# B&R Automation Studio project Panasonic_LinkaPowerCP2_A2021055 (part 3)

### Config.mprecipexml - 5PC900_TS17_00/mappServices/Config.mprecipexml
```
Element gRemPremenneP1 (Type=mprecipexml)
```

### Config_1.mprecipexml - 5PC900_TS17_00/mappServices/Config_1.mprecipexml
```
Element gRemPremenneP2 (Type=mprecipexml)
```

### Config_2.mprecipexml - 5PC900_TS17_00/mappServices/Config_2.mprecipexml
```
Element gRemPremenneP34 (Type=mprecipexml)
```

### Config_3.mpalarmxhistory - 5PC900_TS17_00/mappServices/Config_3.mpalarmxhistory
```
Element gAlarmXHistory (Type=mpalarmxhistory)
  mapp.AlarmX.History:
    Export:
      FileNamePattern = Alarms_%d_%m_%Y_%H_%M_%S.csv
      TimeStampPattern = %d-%m-%Y %H:%M:%S:%L
```

### Config_4.mpalarmxcore - 5PC900_TS17_00/mappServices/Config_4.mpalarmxcore
```
Element gAlarmXCore (Type=mpalarmxcore)
  mapp.AlarmX.Core.Configuration:
    [0]:
      Name = A100
      Message = ST1_Vytah - paletka na vystupe dopravnika vytahu !!!
      Code = 100
      Behavior = PersistentAlarm
    [1]:
      Name = A101
      Message = ST1_Vytah - narusenie optickej bariery !!!
      Code = 101
      Behavior = PersistentAlarm
    [2]:
      Name = A102
      Message = ST1_Vytah - porucha navezenia paletky na dopravnik vytahu !!!
      Code = 102
      Behavior = PersistentAlarm
    [3]:
      Name = A103
      Message = ST1_Vytah - porucha precitania kodu paletky !!!
      Code = 103
      Behavior = PersistentAlarm
    [4]:
      Name = A104
      Message = ST1_Vytah - porucha komunikacie zo serverom !!!
      Code = 104
      Behavior = PersistentAlarm
    [5]:
      Name = A105
      Message = ST1_Vytah - porucha odoslania fotiek na server !!!
      Code = 105
      Behavior = PersistentAlarm
    [6]:
      Name = A106
      Message = ST1_Vytah - CAM 2 porucha komunikacie FTP !!!
      Code = 106
      Behavior = PersistentAlarm
    [7]:
      Name = A107
      Message = ST1_Vytah - CAM 3 porucha komunikacie FTP !!!
      Code = 107
      Behavior = PersistentAlarm
    [8]:
      Name = A108
      Message = ST1_Vytah - CAM 4 porucha komunikacie FTP !!!
      Code = 108
      Behavior = PersistentAlarm
    [9]:
      Name = A109
      Message = ST1_Vytah - CAM 5 porucha komunikacie FTP !!!
      Code = 109
      Behavior = PersistentAlarm
    [10]:
      Name = A110
      Message = ST1_Vytah - porucha serva zdvihu vytahu !!!
      Code = 110
      Behavior = PersistentAlarm
    [11]:
      Name = A111
      Message = ST2_Srobovanie - porucha vysunutia centrovacky !!!
      Code = 111
      Behavior = PersistentAlarm
    [12]:
      Name = A112
      Message = ST2_Srobovanie - porucha zasunutia centrovacky !!!
      Code = 112
      Behavior = PersistentAlarm
    [13]:
      Name = A113
      Message = ST2_Srobovanie - porucha precitania kodu paletky !!!
      Code = 113
      Behavior = PersistentAlarm
    [14]:
      Name = A114
      Message = ST2_Srobovanie - porucha komunikacie zo serverom !!!
      Code = 114
      Behavior = PersistentAlarm
    [15]:
      Name = A115
      Message = ST2_Srobovanie - porucha odoslania fotiek na server !!!
      Code = 115
      Behavior = PersistentAlarm
    [16]:
      Name = A116
      Message = ST2_Srobovanie - CAM 6 porucha komunikacie FTP !!!
      Code = 116
      Behavior = PersistentAlarm
    [17]:
      Name = A117
      Message = ST2_Srobovanie - porucha serva manipulatora os X !!!
      Code = 117
      Behavior = PersistentAlarm
    [18]:
      Name = A118
      Message = ST2_Srobovanie - porucha serva manipulatora os Y !!!
      Code = 118
      Behavior = PersistentAlarm
    [19]:
      Name = A119
      Message = ST2_Srobovanie - skrutka K30 nieje pripravena !!!
      Code = 119
      Behavior = PersistentAlarm
    [20]:
      Name = A120
      Message = ST2_Srobovanie - skrutka M5 nieje pripravena !!!
      Code = 120
      Behavior = PersistentAlarm
    [21]:
      Name = A121
      Message = ST2_Srobovanie - skrutka M4 nieje pripravena !!!
      Code = 121
      Behavior = PersistentAlarm
    [22]:
      Name = A122
      Message = P1_Robot - porucha napajania !!!
      Code = 122
      Behavior = PersistentAlarm
    [23]:
      Name = A123
      Message = P1_Robot - nieje online !!!
      Code = 123
      Behavior = PersistentAlarm
    [24]:
      Name = A124
      Message = Pracovisko 1 - Porucha tlaku vzduchu !!!
      Code = 124
      Behavior = PersistentAlarm
    [25]:
      Name = A125
      Message = Pracovisko 1 - Moduly IO niesu online !!!
      Code = 125
      Behavior = PersistentAlarm
    [26]:
      Name = A126
      Message = ST2_Srobovanie - porucha serva manipulatora os Z M4 !!!
      Code = 126
      Behavior = PersistentAlarm
    [27]:
      Name = A127
      Message = ST2_Srobovanie - porucha serva manipulatora os Z M5 !!!
      Code = 127
      Behavior = PersistentAlarm
    [28]:
      Name = A128
      Message = Pracovisko 1 - Porucha skrutkovacieho setu M4 !!!
      Code = 128
      Behavior = PersistentAlarm
    [29]:
      Name = A129
      Message = Pracovisko 1 - Porucha skrutkovacieho setu M5 !!!
      Code = 129
      Behavior = PersistentAlarm
    [30]:
      Name = A130
      Message = Pracovisko 1 - Narusenie optickej bariery na vystupe bunky !!!
      Code = 130
      Behavior = PersistentAlarm
    [31]:
      Name = A131
      Message = Pracovisko 1 - Modul DS12 nieje online !!!
      Code = 131
      Behavior = PersistentAlarm
    [32]:
      Name = A132
      Message = Pracovisko 1 - Modul SI11 nieje online !!!
      Code = 132
      Behavior = PersistentAlarm
    [33]:
      Name = A133
      Message = Pracovisko 1 - Modul SI12 nieje online !!!
      Code = 133
      Behavior = PersistentAlarm
    [34]:
      Name = A134
      Message = Pracovisko 1 - Ventilovy termnal Bunky 1 nieje online !!!
      Code = 134
      Behavior = PersistentAlarm
    [35]:
      Name = A135
      Message = Pracovisko 1 - Ventilovy termnal VT5 nieje online !!!
      Code = 135
      Behavior = PersistentAlarm
    [36]:
      Name = A136
      Message = ST2_Srobovanie - Skrutkovacka K30 nieje online !!!
      Code = 136
      Behavior = PersistentAlarm
    [37]:
      Name = A137
      Message = ST2_Srobovanie - Skrutkovacka M5 nieje online !!!
      Code = 137
      Behavior = PersistentAlarm
    [38]:
      Name = A138
      Message = ST2_Srobovanie - Skrutkovacka M4 nieje online !!!
      Code = 138
      Behavior = PersistentAlarm
    [39]:
      Name = A139
      Message = Pracovisko 1 - Kamery KAM2, KAM4 a KAM6 niesu online !!!
      Code = 139
      Behavior = PersistentAlarm
    [40]:
      Name = A140
      Message = Pracovisko 1 - Kamera KAM3 nieje online !!!
      Code = 140
      Behavior = PersistentAlarm
    [41]:
      Name = A141
      Message = Pracovisko 1 - Kamera KAM5 nieje online !!!
      Code = 141
      Behavior = PersistentAlarm
    [42]:
      Name = A142
      Message = ST2_Srobovanie - Porucha vysunutia skrutkovacky K30 !!!
      Code = 142
      Behavior = PersistentAlarm
    [43]:
      Name = A143
      Message = ST2_Srobovanie - Porucha vysunutia skrutkovacky M5  !!!
      Code = 143
      Behavior = PersistentAlarm
    [44]:
      Name = A144
      Message = ST2_Srobovanie - Porucha vysunutia skrutkovacky M4 !!!
      Code = 144
      Behavior = PersistentAlarm
    [45]:
      Name = A145
      Message = P1_Robot - porucha !!!
      Code = 145
      Behavior = PersistentAlarm
    [46]:
      Name = A146
      Message = ST2_Srobovanie - Presiahnuty cas skrutkovania skrutky K30 !!!
      Code = 146
      Behavior = PersistentAlarm
    [47]:
      Name = A147
      Message = ST2_Srobovanie - Presiahnuty cas skrutkovania skrutky M5 !!!
      Code = 147
      Behavior = PersistentAlarm
    [48]:
      Name = A148
      Message = ST2_Srobovanie - Presiahnuty cas skrutkovania skrutky M4 !!!
      Code = 148
      Behavior = PersistentAlarm
    [49]:
      Name = A149
      Message = ST2_Srobovanie - Skrutkovacka K30 nieje READY !!!
      Code = 149
      Behavior = PersistentAlarm
    [50]:
      Name = A150
      Message = ST2_Srobovanie - Skrutkovacka M5 nieje READY !!!
      Code = 150
      Behavior = PersistentAlarm
    [51]:
      Name = A151
      Message = ST2_Srobovanie - Skrutkovacka M4 nieje READY !!!
      Code = 151
      Behavior = PersistentAlarm
    [52]:
      Name = A152
      Message = Pracovisko 1 - Prekrocena teplota motora vrchneho dopravnika !!!
      Code = 152
      Behavior = PersistentAlarm
    [53]:
      Name = A153
      Message = Pracovisko 1 - Prekrocena teplota motora spodneho dopravnika !!!
      Code = 153
      Behavior = PersistentAlarm
    [54]:
      Name = A154
      Message = Pracovisko 1 - Narusenie optickej bariery na vstupe bunky !!!
      Code = 154
      Behavior = PersistentAlarm
    [55]:
      Name = A155
      Message = ST1_Vytah - Prekrocena teplota motora dopravnika !!!
      Code = 155
      Behavior = PersistentAlarm
    [56]:
      Name = A156
      Message = Pracovisko 1 - Bolo stlacene tlacitko CS na ovladacom paneli !!!
      Code = 156
      Behavior = PersistentAlarm
    [57]:
      Name = A157
      Message = Pracovisko 1 - Bolo stlacene tlacitko CS na rozvodnej skrini !!!
      Code = 157
      Behavior = PersistentAlarm
    [58]:
      Name = A158
      Message = Pracovisko 1 - Bolo stlacene tlacitko CS robota !!!
      Code = 158
      Behavior = PersistentAlarm
    [59]:
      Name = A159
      Message = P1_Robot - Porucha odobratia foamov z paletky !!!
      Code = 159
      Behavior = PersistentAlarm
    [60]:
      Name = A160
      Message = P1_Robot - Porucha odobratia busbarov z paletky !!!
      Code = 160
      Behavior = PersistentAlarm
    [61]:
      Name = A161
      Message = ST2_Srobovanie - Porucha vyvezenia paletky zo stopra !!!
      Code = 161
      Behavior = PersistentAlarm
    [62]:
      Name = A162
      Message = P1_Akumulacny stoper - Porucha vyvezenia paletky zo stopra !!!
      Code = 162
      Behavior = PersistentAlarm
    [63]:
      Name = A163
      Message = P1_Spodny stoper - Porucha vyvezenia paletky zo stopra !!!
      Code = 163
      Behavior = PersistentAlarm
    [64]:
      Name = A164
      Message = ST1_Vytah - Porucha komunikacie s kamerou CAM 2 !!!
      Code = 164
      Behavior = PersistentAlarm
    [65]:
      Name = A165
      Message = ST1_Vytah - Porucha komunikacie s kamerou CAM 5 !!!
      Code = 165
      Behavior = PersistentAlarm
    [66]:
      Name = A166
      Message = ST1_Vytah - Porucha komunikacie s kamerou CAM 4 !!!
      Code = 166
      Behavior = PersistentAlarm
    [67]:
      Name = A167
      Message = ST1_Vytah - Porucha komunikacie s kamerou CAM 3 !!!
      Code = 167
      Behavior = PersistentAlarm
    [68]:
      Name = A168
      Message = ST2_Srobovanie - Porucha komunikacie s kamerou CAM 6 !!!
      Code = 168
      Behavior = PersistentAlarm
    [69]:
      Name = A200
      Message = ST3_Zakladanie tesnenia - porucha precitania kodu paletky !!!
      Code = 200
      Behavior = PersistentAlarm
    [70]:
      Name = A201
      Message = ST3_Zakladanie tesnenia - porucha precitania QR kodu !!!
      Code = 201
      Behavior = PersistentAlarm
    [71]:
      Name = A202
      Message = ST3_Zakladanie tesnenia - porucha serva zdvihu !!!
      Code = 202
      Behavior = PersistentAlarm
    [72]:
      Name = A203
      Message = ST3_Zakladanie tesnenia - porucha serva pojazdu !!!
      Code = 203
      Behavior = PersistentAlarm
    [73]:
      Name = A204
      Message = ST3_Zakladanie tesnenia - porucha vysunutia pritlacania !!!
      Code = 204
      Behavior = PersistentAlarm
    [74]:
      Name = A205
      Message = ST3_Zakladanie tesnenia - porucha zasunutia pritlacania !!!
      Code = 205
      Behavior = PersistentAlarm
    [75]:
      Name = A206
      Message = ST3_Zakladanie tesnenia - narusenie optickej bariery !!!
      Code = 206
      Behavior = PersistentAlarm
    [76]:
      Name = A207
      Message = ST3_Zakladanie tesnenia - bol stlaceny bumper suflika !!!
      Code = 207
      Behavior = PersistentAlarm
    [77]:
      Name = A208
      Message = ST3_Zakladanie tesnenia - porucha snimaca kopita IS7 !!!
      Code = 208
      Behavior = PersistentAlarm
    [78]:
      Name = A209
      Message = ST4_Maticovacka - porucha vysunutia centrovacky !!!
      Code = 209
      Behavior = PersistentAlarm
    [79]:
      Name = A210
      Message = ST4_Maticovacka - porucha zasunutia centrovacky !!!
      Code = 210
      Behavior = PersistentAlarm
    [80]:
      Name = A211
      Message = ST4_Maticovacka - porucha precitania kodu paletky !!!
      Code = 211
      Behavior = PersistentAlarm
    [81]:
      Name = A212
      Message = ST5_Srobovanie - porucha vysunutia centrovacky !!!
      Code = 212
      Behavior = PersistentAlarm
    [82]:
      Name = A213
      Message = ST5_Srobovanie - porucha zasunutia centrovacky !!!
      Code = 213
      Behavior = PersistentAlarm
    [83]:
      Name = A214
      Message = ST5_Srobovanie - porucha precitania kodu paletky !!!
      Code = 214
      Behavior = PersistentAlarm
    [84]:
      Name = A215
      Message = ST5_Srobovanie - porucha serva manipulatora os X !!!
      Code = 215
      Behavior = PersistentAlarm
    [85]:
      Name = A216
      Message = ST5_Srobovanie - porucha serva manipulatora os Y !!!
      Code = 216
      Behavior = PersistentAlarm
    [86]:
      Name = A217
      Message = ST6_Zvaranie - porucha vysunutia centrovacky !!!
      Code = 217
      Behavior = PersistentAlarm
    [87]:
      Name = A218
      Message = ST6_Zvaranie - porucha zasunutia centrovacky !!!
      Code = 218
      Behavior = PersistentAlarm
    [88]:
      Name = A219
      Message = ST6_Zvaranie - porucha precitania kodu paletky !!!
      Code = 219
      Behavior = PersistentAlarm
    [89]:
      Name = A220
      Message = ST6_Zvaranie - porucha serva zdvihu zvarania !!!
      Code = 220
      Behavior = PersistentAlarm
    [90]:
      Name = A221
      Message = ST6_Zvaranie - porucha presunu pojazdu zvarania !!!
      Code = 221
      Behavior = PersistentAlarm
    [91]:
      Name = A222
      Message = ST6_Zvaranie - porucha zvaracky !!!
      Code = 222
      Behavior = PersistentAlarm
    [92]:
      Name = A223
      Message = ST6_Cistenie - porucha zatvorenia dveri !!!
      Code = 223
      Behavior = PersistentAlarm
    [93]:
      Name = A224
      Message = ST6_Cistenie - porucha otvorenia dveri !!!
      Code = 224
      Behavior = PersistentAlarm
    [94]:
      Name = A225
      Message = ST3_Zakladanie tesnenia - CAM 1 porucha komunikacie FTP !!!
      Code = 225
      Behavior = PersistentAlarm
    [95]:
      Name = A226
      Message = ST3_Zakladanie tesnenia - CAM 7 porucha komunikacie FTP !!!
      Code = 226
      Behavior = PersistentAlarm
    [96]:
      Name = A227
      Message = ST3_Zakladanie tesnenia - CAM 8 porucha komunikacie FTP !!!
      Code = 227
      Behavior = PersistentAlarm
    [97]:
      Name = A228
      Message = ST3_Zakladanie tesnenia - CAM 17 porucha komunikacie FTP !!!
      Code = 228
      Behavior = PersistentAlarm
    [98]:
      Name = A229
      Message = ST4_Maticovacka - CAM 9 porucha komunikacie FTP !!!
      Code = 229
      Behavior = PersistentAlarm
    [99]:
      Name = A230
      Message = ST3_Zakladanie tesnenia - porucha komunikacie zo serverom !!!
      Code = 230
      Behavior = PersistentAlarm
    [100]:
      Name = A231
      Message = ST4_Maticovacka - porucha komunikacie zo serverom !!!
      Code = 231
      Behavior = PersistentAlarm
    [101]:
      Name = A232
      Message = ST5_Srobovanie - CAM 10 porucha komunikacie FTP !!!
      Code = 232
      Behavior = PersistentAlarm
    [102]:
      Name = A233
      Message = ST5_Srobovanie - porucha komunikacie zo serverom !!!
      Code = 233
      Behavior = PersistentAlarm
    [103]:
      Name = A234
      Message = ST6_Zvaranie - CAM 11 porucha komunikacie FTP !!!
      Code = 234
      Behavior = PersistentAlarm
    [104]:
      Name = A235
      Message = ST6_Zvaranie - CAM 12 porucha komunikacie FTP !!!
      Code = 235
      Behavior = PersistentAlarm
    [105]:
      Name = A236
      Message = ST6_Zvaranie - porucha komunikacie zo serverom !!!
      Code = 236
      Behavior = PersistentAlarm
    [106]:
      Name = A237
      Message = ST5_Srobovanie - skrutka M4 nieje pripravena !!!
      Code = 237
      Behavior = PersistentAlarm
    [107]:
      Name = A238
      Message = ST5_Srobovanie - skrutka M5 nieje pripravena !!!
      Code = 238
      Behavior = PersistentAlarm
    [108]:
      Name = A239
      Message = ST5_Srobovanie - skrutka M6 nieje pripravena !!!
      Code = 239
      Behavior = PersistentAlarm
    [109]:
      Name = A240
      Message = ST4_Maticovacka - matica M4 nieje pripravena !!!
      Code = 240
      Behavior = PersistentAlarm
    [110]:
      Name = A241
      Message = ST5_Srobovanie - porucha serva manipulatora os X !!!
      Code = 241
      Behavior = PersistentAlarm
    [111]:
      Name = A242
      Message = ST5_Srobovanie - porucha serva manipulatora os Y !!!
      Code = 242
      Behavior = PersistentAlarm
    [112]:
      Name = A243
      Message = P2_Robot - porucha napajania !!!
      Code = 243
      Behavior = PersistentAlarm
    [113]:
      Name = A244
      Message = P2_Robot - nieje online !!!
      Code = 244
      Behavior = PersistentAlarm
    [114]:
      Name = A245
      Message = Pracovisko 2 - Porucha tlaku vzduchu !!!
      Code = 245
      Behavior = PersistentAlarm
    [115]:
      Name = A246
      Message = Pracovisko 2 - Moduly IO niesu online !!!
      Code = 246
      Behavior = PersistentAlarm
    [116]:
      Name = A247
      Message = ST5_Srobovanie - porucha serva manipulatora os Z M4 !!!
      Code = 247
      Behavior = PersistentAlarm
    [117]:
      Name = A248
      Message = Pracovisko 2 - Porucha skrutkovacieho setu M4 !!!
      Code = 248
      Behavior = PersistentAlarm
    [118]:
      Name = A249
      Message = Pracovisko 2 - Porucha skrutkovacieho setu matice M4 !!!
      Code = 249
    [119]:
      Name = A250
      Message = Pracovisko 2 - Porucha komunikacie s Panatrace !!!
      Code = 250
      Behavior = PersistentAlarm
    [120]:
      Name = A251
      Message = Pracovisko 2 - Modul DM21 nieje online !!!
      Code = 251
    [121]:
      Name = A252
      Message = Pracovisko 2 - Modul DS21 nieje online !!!
      Code = 252
      Behavior = PersistentAlarm
    [122]:
      Name = A253
      Message = Pracovisko 2 - Modul DS22 nieje online !!!
      Code = 253
      Behavior = PersistentAlarm
    [123]:
      Name = A254
      Message = Pracovisko 2 - Modul DS23 nieje online !!!
      Code = 254
      Behavior = PersistentAlarm
    [124]:
      Name = A255
      Message = Pracovisko 2 - Modul SI21 nieje online !!!
      Code = 255
      Behavior = PersistentAlarm
    [125]:
      Name = A256
      Message = Pracovisko 2 - Modul SI22 nieje online !!!
      Code = 256
      Behavior = PersistentAlarm
    [126]:
      Name = A257
      Message = Pracovisko 2 - Ventilovy termnal Bunky 2 nieje online !!!
      Code = 257
      Behavior = PersistentAlarm
    [127]:
      Name = A258
      Message = Pracovisko 2 - Ventilovy termnal VT2 nieje online !!!
      Code = 258
      Behavior = PersistentAlarm
    [128]:
      Name = A259
      Message = Pracovisko 2 - Ventilovy termnal VT3 nieje online !!!
      Code = 259
      Behavior = PersistentAlarm
    [129]:
      Name = A260
      Message = ST5_Srobovanie - Skrutkovacka M4 nieje online !!!
      Code = 260
      Behavior = PersistentAlarm
    [130]:
      Name = A261
      Message = ST5_Srobovanie - Skrutkovacka M5 nieje online !!!
      Code = 261
      Behavior = PersistentAlarm
    [131]:
      Name = A262
      Message = ST5_Srobovanie - Skrutkovacka M6 nieje online !!!
      Code = 262
      Behavior = PersistentAlarm
    [132]:
      Name = A263
      Message = ST4_Maticovacka - Maticovacka M4 nieje online !!!
      Code = 263
      Behavior = PersistentAlarm
    [133]:
      Name = A264
      Message = Pracovisko 2 - Kamery KAM1, KAM7, KAM10, KAM11, KAM12 a KAM17 niesu online !!!
      Code = 264
      Behavior = PersistentAlarm
    [134]:
      Name = A265
      Message = Pracovisko 2 - Kamera KAM8 nieje online !!!
      Code = 265
      Behavior = PersistentAlarm
    [135]:
      Name = A266
      Message = Pracovisko 2 - Kamera KAM9 nieje online !!!
      Code = 266
      Behavior = PersistentAlarm
    [136]:
      Name = A267
      Message = ST4_Maticovacka - Porucha maticovacky M4 !!!
      Code = 267
      Behavior = PersistentAlarm
    [137]:
      Name = A268
      Message = ST5_Srobovanie - Porucha vysunutia skrutkovacky M4 !!!
      Code = 268
      Behavior = PersistentAlarm
    [138]:
      Name = A269
      Message = ST5_Srobovanie - Porucha vysunutia skrutkovacky M5 !!!
      Code = 269
      Behavior = PersistentAlarm
    [139]:
      Name = A270
      Message = ST5_Srobovanie - Porucha vysunutia skrutkovacky M6 !!!
      Code = 270
      Behavior = PersistentAlarm
    [140]:
      Name = A271
      Message = P2_Robot - porucha !!!
      Code = 271
      Behavior = PersistentAlarm
    [141]:
      Name = A272
      Message = ST5_Srobovanie - Presiahnuty cas skrutkovania skrutky M4 !!!
      Code = 272
      Behavior = PersistentAlarm
    [142]:
      Name = A273
      Message = ST5_Srobovanie - Presiahnuty cas skrutkovania skrutky M5 !!!
      Code = 273
      Behavior = PersistentAlarm
    [143]:
      Name = A274
      Message = ST5_Srobovanie - Presiahnuty cas skrutkovania skrutky M6 !!!
      Code = 274
      Behavior = PersistentAlarm
    [144]:
      Name = A275
      Message = ST5_Srobovanie - Skrutkovacka M4 nieje READY !!!
      Code = 275
      Behavior = PersistentAlarm
    [145]:
      Name = A276
      Message = ST5_Srobovanie - Skrutkovacka M5 nieje READY !!!
      Code = 276
      Behavior = PersistentAlarm
    [146]:
      Name = A277
      Message = ST5_Srobovanie - Skrutkovacka M6 nieje READY !!!
      Code = 277
      Behavior = PersistentAlarm
    [147]:
      Name = A278
      Message = Pracovisko 2 - Prekrocena teplota motora vrchneho dopravnika !!!
      Code = 278
      Behavior = PersistentAlarm
    [148]:
      Name = A279
      Message = Pracovisko 2 - Prekrocena teplota motora spodneho dopravnika !!!
      Code = 279
      Behavior = PersistentAlarm
    [149]:
      Name = A280
      Message = Pracovisko 2 - Narusenie optickej bariery na vystupe !!!
      Code = 280
      Behavior = PersistentAlarm
    [150]:
      Name = A281
      Message = Pracovisko 2 - Bolo stlacene tlacitko CS na ovladacom paneli !!!
      Code = 281
      Behavior = PersistentAlarm
    [151]:
      Name = A282
      Message = Pracovisko 2 - Bolo stlacene tlacitko CS na rozvodnej skrini !!!
      Code = 282
      Behavior = PersistentAlarm
    [152]:
      Name = A283
      Message = Pracovisko 2 - Bolo stlacene tlacitko CS robota !!!
      Code = 283
      Behavior = PersistentAlarm
    [153]:
      Name = A284
      Message = Pracovisko 2 - Bolo stlacene tlacitko CS na dvojrucnom ovladani !!!
      Code = 284
      Behavior = PersistentAlarm
    [154]:
      Name = A285
      Message = P2_Robot - Porucha odobratia Top Coveru z paletky !!!
      Code = 285
      Behavior = PersistentAlarm
    [155]:
      Name = A286
      Message = ST3_Zakladanie tesnenia - Porucha vyvezenia paletky zo stopra !!!
      Code = 286
      Behavior = PersistentAlarm
    [156]:
      Name = A287
      Message = ST4_Maticovacka - Porucha vyvezenia paletky zo stopra !!!
      Code = 287
      Behavior = PersistentAlarm
    [157]:
      Name = A288
      Message = ST5_Srobovanie - Porucha vyvezenia paletky zo stopra !!!
      Code = 288
      Behavior = PersistentAlarm
    [158]:
      Name = A289
      Message = ST6_Zvaranie - Porucha vyvezenia paletky zo stopra !!!
      Code = 289
      Behavior = PersistentAlarm
    [159]:
      Name = A290
      Message = ST3_Zakladanie tesnenia - Porucha komunikacie s kamerou CAM 1 !!!
      Code = 290
    [160]:
      Name = A291
      Message = ST3_Zakladanie tesnenia - Porucha komunikacie s kamerou CAM 7 !!!
      Code = 291
      Behavior = PersistentAlarm
    [161]:
      Name = A292
      Message = ST3_Zakladanie tesnenia - Porucha komunikacie s kamerou CAM 8 !!!
      Code = 292
      Behavior = PersistentAlarm
    [162]:
      Name = A293
      Message = ST3_Zakladanie tesnenia - Porucha komunikacie s kamerou CAM 17 !!!
      Code = 293
      Behavior = PersistentAlarm
    [163]:
      Name = A294
      Message = ST4_Maticovacka - Porucha komunikacie s kamerou CAM 9 !!!
      Code = 294
      Behavior = PersistentAlarm
    [164]:
      Name = A295
      Message = ST5_Srobovanie - Porucha komunikacie s kamerou CAM 10 !!!
      Code = 295
      Behavior = PersistentAlarm
    [165]:
      Name = A296
      Message = ST6_Zvaranie - Porucha komunikacie s kamerou CAM 11 !!!
      Code = 296
      Behavior = PersistentAlarm
    [166]:
      Name = A297
      Message = ST6_Zvaranie - Porucha komunikacie s kamerou CAM 12 !!!
      Code = 297
      Behavior = PersistentAlarm
    [167]:
      Name = A298
      Message = ST4_Maticovacka - Porucha pripravy matice M4 !!!
      Code = 298
      Behavior = PersistentAlarm
    [168]:
      Name = A299
      Message = Akumulacny stoper - Porucha vyvezenia paletky zo stopra !!!
      Code = 299
      Behavior = PersistentAlarm
    [169]:
      Name = A300
      Message = ST7_Srobovanie - porucha vysunutia centrovacky !!!
      Code = 300
      Behavior = PersistentAlarm
    [170]:
      Name = A301
      Message = ST7_Srobovanie - porucha zasunutia centrovacky !!!
      Code = 301
      Behavior = PersistentAlarm
    [171]:
      Name = A302
      Message = ST8A_Leakage test A - porucha vysunutia centrovacky !!!
      Code = 302
      Behavior = PersistentAlarm
    [172]:
      Name = A303
      Message = ST8A_Leakage test A - porucha zasunutia centrovacky !!!
      Code = 303
      Behavior = PersistentAlarm
    [173]:
      Name = A304
      Message = ST8B_Leakage test B - porucha vysunutia centrovacky !!!
      Code = 304
      Behavior = PersistentAlarm
    [174]:
      Name = A305
      Message = ST8B_Leakage test B - porucha zasunutia centrovacky !!!
      Code = 305
      Behavior = PersistentAlarm
    [175]:
      Name = A306
      Message = ST8A_Leakage test A - porucha vysunutia pritlaku !!!
      Code = 306
      Behavior = PersistentAlarm
    [176]:
      Name = A307
      Message = ST8A_Leakage test A - porucha zasunutia pritlaku !!!
      Code = 307
      Behavior = PersistentAlarm
    [177]:
      Name = A308
      Message = ST8B_Leakage test B - porucha vysunutia pritlaku !!!
      Code = 308
      Behavior = PersistentAlarm
    [178]:
      Name = A309
      Message = ST8B_Leakage test B - porucha zasunutia pritlaku !!!
      Code = 309
      Behavior = PersistentAlarm
    [179]:
      Name = A310
      Message = ST8A_Leakage test A - porucha precitania kodu paletky !!!
      Code = 310
      Behavior = PersistentAlarm
    [180]:
      Name = A311
      Message = ST8A_Leakage test A - porucha komunikacie zo serverom !!!
      Code = 311
      Behavior = PersistentAlarm
    [181]:
      Name = A312
      Message = ST8B_Leakage test B - porucha precitania kodu paletky !!!
      Code = 312
      Behavior = PersistentAlarm
    [182]:
      Name = A313
      Message = ST8B_Leakage test B - porucha komunikacie zo serverom !!!
      Code = 313
      Behavior = PersistentAlarm
    [183]:
      Name = A314
      Message = ST8A_Leakage test A - je zalozeny nespravny typ spodneho kopita !!!
      Code = 314
      Behavior = PersistentAlarm
    [184]:
      Name = A315
      Message = ST8B_Leakage test B - je zalozeny nespravny typ spodneho kopita !!!
      Code = 315
      Behavior = PersistentAlarm
    [185]:
      Name = A316
      Message = ST7_Srobovanie - porucha vysunutia kontaktov HV testu !!!
      Code = 316
      Behavior = PersistentAlarm
    [186]:
      Name = A317
      Message = ST7_Srobovanie - porucha zasunutia kontaktov HV testu !!!
      Code = 317
      Behavior = PersistentAlarm
    [187]:
      Name = A318
      Message = ST7_Srobovanie - porucha vysunutia HV testu !!!
      Code = 318
      Behavior = PersistentAlarm
    [188]:
      Name = A319
      Message = ST7_Srobovanie - porucha zasunutia HV testu !!!
      Code = 319
      Behavior = PersistentAlarm
    [189]:
      Name = A320
      Message = ST7_Srobovanie - CAM 13 porucha komunikacie FTP !!!
      Code = 320
      Behavior = PersistentAlarm
    [190]:
      Name = A321
      Message = ST7_Srobovanie - porucha precitania kodu paletky !!!
      Code = 321
      Behavior = PersistentAlarm
    [191]:
      Name = A322
      Message = ST7_Srobovanie - porucha serva manipulatora os Y !!!
      Code = 322
      Behavior = PersistentAlarm
    [192]:
      Name = A323
      Message = Pracovisko 3 - Porucha tlaku vzduchu !!!
      Code = 323
      Behavior = PersistentAlarm
    [193]:
      Name = A324
      Message = ST7_Srobovanie - Skrutkovacka M5 nieje online !!!
      Code = 324
      Behavior = PersistentAlarm
    [194]:
      Name = A325
      Message = ST7_Srobovanie - porucha komunikacie zo serverom !!!
      Code = 325
      Behavior = PersistentAlarm
    [195]:
      Name = A326
      Message = ST7_HV Test - je zalozeny nespravny typ spodneho kopita !!!
      Code = 326
      Behavior = PersistentAlarm
    [196]:
      Name = A327
      Message = ST7_Srobovanie - skrutka M5 nieje pripravena !!!
      Code = 327
      Behavior = PersistentAlarm
    [197]:
      Name = A328
      Message = ST7_Srobovanie - skrutka K40 nieje pripravena !!!
      Code = 328
      Behavior = PersistentAlarm
    [198]:
      Name = A329
      Message = ST7_Srobovanie - Skrutkovacka K40 nieje online !!!
      Code = 329
      Behavior = PersistentAlarm
    [199]:
      Name = A330
      Message = ST7_Srobovanie - Kamera KAM13 nieje online !!!
      Code = 330
      Behavior = PersistentAlarm
    [200]:
      Name = A331
      Message = Pracovisko 3 - Moduly IO niesu online !!!
      Code = 331
      Behavior = PersistentAlarm
    [201]:
      Name = A332
      Message = ST7_Srobovanie - porucha serva manipulatora os Z M5 !!!
      Code = 332
      Behavior = PersistentAlarm
    [202]:
      Name = A333
      Message = Pracovisko 3 - Modul DI33 nieje online !!!
      Code = 333
      Behavior = PersistentAlarm
    [203]:
      Name = A334
      Message = Pracovisko 3 - Porucha skrutkovacieho setu M5 !!!
      Code = 334
      Behavior = PersistentAlarm
    [204]:
      Name = A335
      Message = Pracovisko 3 - Prekrocena teplota motora zadneho vrchneho dopravnika !!!
      Code = 335
      Behavior = PersistentAlarm
    [205]:
      Name = A336
      Message = Pracovisko 3 - Prekrocena teplota motora prveho priecneho dopravnika !!!
      Code = 336
      Behavior = PersistentAlarm
    [206]:
      Name = A337
      Message = Pracovisko 3 - Prekrocena teplota motora druheho priecneho dopravnika !!!
      Code = 337
      Behavior = PersistentAlarm
    [207]:
      Name = A338
      Message = Pracovisko 3 - Modul DS33 nieje online !!!
      Code = 338
      Behavior = PersistentAlarm
    [208]:
      Name = A339
      Message = Pracovisko 3 - Modul SI31 nieje online !!!
      Code = 339
      Behavior = PersistentAlarm
    [209]:
      Name = A340
      Message = Pracovisko 3 - Ventilovy termnal Bunky 3 nieje online !!!
      Code = 340
      Behavior = PersistentAlarm
    [210]:
      Name = A341
      Message = Pracovisko 3 - Ventilovy termnal VT7 nieje online !!!
      Code = 341
      Behavior = PersistentAlarm
    [211]:
      Name = A342
      Message = ST7_Srobovanie - Porucha vysunutia skrutkovacky K40 !!!
      Code = 342
      Behavior = PersistentAlarm
    [212]:
      Name = A343
      Message = ST7_Srobovanie - Porucha vysunutia skrutkovacky M5 !!!
      Code = 343
      Behavior = PersistentAlarm
    [213]:
      Name = A344
      Message = ST7_Srobovanie - Skrutkovacka K40 nieje READY !!!
      Code = 344
      Behavior = PersistentAlarm
    [214]:
      Name = A345
      Message = ST7_Srobovanie - Skrutkovacka M5 nieje READY !!!
      Code = 345
      Behavior = PersistentAlarm
    [215]:
      Name = A346
      Message = ST7_Srobovanie - Presiahnuty cas skrutkovania skrutky K40 !!!
      Code = 346
      Behavior = PersistentAlarm
    [216]:
      Name = A347
      Message = ST7_Srobovanie - Presiahnuty cas skrutkovania skrutky M5 !!!
      Code = 347
      Behavior = PersistentAlarm
    [217]:
      Name = A348
      Message = Pracovisko 3 - Prekrocena teplota motora predneho vrchneho dopravnika !!!
      Code = 348
      Behavior = PersistentAlarm
    [218]:
      Name = A349
      Message = Pracovisko 3 - Prekrocena teplota motora spodneho dopravnika !!!
      Code = 349
      Behavior = PersistentAlarm
    [219]:
      Name = A350
      Message = Pracovisko 3 - Narusenie optickej bariery na vstupe !!!
      Code = 350
      Behavior = PersistentAlarm
    [220]:
      Name = A351
      Message = Pracovisko 3 - Narusenie optickej bariery na vystupe !!!
      Code = 351
      Behavior = PersistentAlarm
    [221]:
      Name = A352
      Message = Pracovisko 3 - Bolo stlacene tlacitko CS na rozvodnej skrini !!!
      Code = 352
      Behavior = PersistentAlarm
    [222]:
      Name = A353
      Message = P3_Spodny stoper - Porucha vyvezenia paletky zo stopra !!!
      Code = 353
      Behavior = PersistentAlarm
    [223]:
      Name = A354
      Message = P3_Vstupny stoper - Porucha vyvezenia paletky zo stopra !!!
      Code = 354
      Behavior = PersistentAlarm
    [224]:
      Name = A355
      Message = ST7_Srobovanie - Porucha vyvezenia paletky zo stopra !!!
      Code = 355
      Behavior = PersistentAlarm
    [225]:
      Name = A356
      Message = P3_Akumulacny stoper - Porucha vyvezenia paletky zo stopra !!!
      Code = 356
      Behavior = PersistentAlarm
    [226]:
      Name = A357
      Message = ST8A_Leakage test A - Porucha vyvezenia paletky zo stopra !!!
      Code = 357
      Behavior = PersistentAlarm
    [227]:
      Name = A358
      Message = ST8B_Leakage test B - Porucha vyvezenia paletky zo stopra !!!
      Code = 358
      Behavior = PersistentAlarm
    [228]:
      Name = A359
      Message = ST7_Srobovanie - Porucha komunikacie s kamerou CAM 13 !!!
      Code = 359
      Behavior = PersistentAlarm
    [229]:
      Name = A360
      Message = ST7_HV Test - Porucha vysunutia centrovacky !!!
      Code = 360
      Behavior = PersistentAlarm
    [230]:
      Name = A361
      Message = ST7_HV Test - Porucha zasunutia centrovacky !!!
      Code = 361
      Behavior = PersistentAlarm
    [231]:
      Name = A362
      Message = ST7_HV Test - Porucha vysunutia spodnych kontaktov !!!
      Code = 362
      Behavior = PersistentAlarm
    [232]:
      Name = A363
      Message = ST7_HV Test - Porucha zasunutia spodnych kontaktov !!!
      Code = 363
      Behavior = PersistentAlarm
    [233]:
      Name = A364
      Message = ST7_HV Test - Porucha vysunutia hornych kontaktov !!!
      Code = 364
    [234]:
      Name = A365
      Message = ST7_HV Test - Porucha zasunutia hornych kontaktov !!!
      Code = 365
      Behavior = PersistentAlarm
    [235]:
      Name = A366
      Message = ST7_HV Test - Porucha precitania kodu paletky !!!
      Code = 366
      Behavior = PersistentAlarm
    [236]:
      Name = A367
      Message = ST7_HV Test - Porucha vyvezenia paletky zo stopra !!!
      Code = 367
      Behavior = PersistentAlarm
    [237]:
      Name = A368
      Message = P3_Zdvizka pred Leakage Testom A - Porucha vysunutia zdvizky !!!
      Code = 368
      Behavior = PersistentAlarm
    [238]:
      Name = A369
      Message = P3_Zdvizka pred Leakage Testom A - Porucha zasunutia zdvizky !!!
      Code = 369
      Behavior = PersistentAlarm
    [239]:
      Name = A370
      Message = P3_Zdvizka pred Leakage Testom A - Porucha strednej polohy zdvizky !!!
      Code = 370
      Behavior = PersistentAlarm
    [240]:
      Name = A371
      Message = P3_Zdvizka pred Leakage Testom B - Porucha vysunutia zdvizky !!!
      Code = 371
      Behavior = PersistentAlarm
    [241]:
      Name = A372
      Message = P3_Zdvizka pred Leakage Testom B - Porucha zasunutia zdvizky !!!
      Code = 372
      Behavior = PersistentAlarm
    [242]:
      Name = A373
      Message = P3_Zdvizka pred Leakage Testom B - Porucha strednej polohy zdvizky !!!
      Code = 373
      Behavior = PersistentAlarm
    [243]:
      Name = A374
      Message = P3_Zdvizka za Leakage Testom A - Porucha vysunutia zdvizky !!!
      Code = 374
      Behavior = PersistentAlarm
    [244]:
      Name = A375
      Message = P3_Zdvizka za Leakage Testom A - Porucha zasunutia zdvizky !!!
      Code = 375
      Behavior = PersistentAlarm
    [245]:
      Name = A376
      Message = P3_Zdvizka za Leakage Testom A - Porucha strednej polohy zdvizky !!!
      Code = 376
      Behavior = PersistentAlarm
    [246]:
      Name = A377
      Message = P3_Zdvizka za Leakage Testom B - Porucha vysunutia zdvizky !!!
      Code = 377
      Behavior = PersistentAlarm
    [247]:
      Name = A378
      Message = P3_Zdvizka za Leakage Testom B - Porucha zasunutia zdvizky !!!
      Code = 378
      Behavior = PersistentAlarm
    [248]:
      Name = A379
      Message = P3_Zdvizka za Leakage Testom B - Porucha strednej polohy zdvizky !!!
      Code = 379
      Behavior = PersistentAlarm
    [249]:
      Name = A400
      Message = ST_Funkcny test A - porucha vysunutia centrovacky !!!
      Code = 400
      Behavior = PersistentAlarm
    [250]:
      Name = A401
      Message = ST_Funkcny test A - porucha zasunutia centrovacky !!!
      Code = 401
      Behavior = PersistentAlarm
    [251]:
      Name = A402
      Message = ST_Funkcny test B - porucha vysunutia centrovacky !!!
      Code = 402
      Behavior = PersistentAlarm
    [252]:
      Name = A403
      Message = ST_Funkcny test B - porucha zasunutia centrovacky !!!
      Code = 403
      Behavior = PersistentAlarm
    [253]:
      Name = A404
      Message = ST9_Etiketovacka - porucha vysunutia centrovacky !!!
      Code = 404
      Behavior = PersistentAlarm
    [254]:
      Name = A405
      Message = ST9_Etiketovacka - porucha zasunutia centrovacky !!!
      Code = 405
      Behavior = PersistentAlarm
    [255]:
      Name = A406
      Message = ST9_Etiketovacka - porucha precitania kodu paletky !!!
      Code = 406
      Behavior = PersistentAlarm
    [256]:
      Name = A407
      Message = Pracovisko 4 - Porucha tlaku vzduchu !!!
      Code = 407
      Behavior = PersistentAlarm
    [257]:
      Name = A408
      Message = ST9_Etiketovacka - porucha serva zdvihu aplikatora etikiet !!!
      Code = 408
      Behavior = PersistentAlarm
    [258]:
      Name = A409
      Message = ST9_Etiketovacka - porucha komunikacie zo serverom !!!
      Code = 409
      Behavior = PersistentAlarm
    [259]:
      Name = A410
      Message = ST10_Vytah - CAM 16 porucha komunikacie FTP !!!
      Code = 410
      Behavior = PersistentAlarm
    [260]:
      Name = A411
      Message = ST10_Vytah - paletka na vystupe dopravnika vytahu !!!
      Code = 411
      Behavior = PersistentAlarm
    [261]:
      Name = A412
      Message = ST10_Vytah - narusenie optickej bariery !!!
      Code = 412
      Behavior = PersistentAlarm
    [262]:
      Name = A413
      Message = Pracovisko 4 - Kamera KAM15 a KAM16 nieje online !!!
      Code = 413
      Behavior = PersistentAlarm
    [263]:
      Name = A414
      Message = Pracovisko 4 - Kamera KAM14 nieje online !!!
      Code = 414
      Behavior = PersistentAlarm
    [264]:
      Name = A415
      Message = ST10_Vytah - porucha komunikacie zo serverom !!!
      Code = 415
      Behavior = PersistentAlarm
    [265]:
      Name = A416
      Message = ST10_Vytah - porucha navezenia paletky na dopravnik vytahu !!!
      Code = 416
      Behavior = PersistentAlarm
    [266]:
      Name = A417
      Message = Pracovisko 4 - Ventilovy termnal VT8 nieje online !!!
      Code = 417
      Behavior = PersistentAlarm
    [267]:
      Name = A418
      Message = ST10_Vytah - porucha precitania kodu paletky !!!
      Code = 418
      Behavior = PersistentAlarm
    [268]:
      Name = A419
      Message = ST_Funkcny test A - porucha vysunutia hornych kontaktov !!!
      Code = 419
      Behavior = PersistentAlarm
    [269]:
      Name = A420
      Message = ST_Funkcny test A - porucha zasunutia hornych kontaktov !!!
      Code = 420
      Behavior = PersistentAlarm
    [270]:
      Name = A421
      Message = ST_Funkcny test A - porucha vysunutia spodnych kontaktov !!!
      Code = 421
      Behavior = PersistentAlarm
    [271]:
      Name = A422
      Message = ST_Funkcny test A - porucha zasunutia spodnych kontaktov !!!
      Code = 422
      Behavior = PersistentAlarm
    [272]:
      Name = A423
      Message = ST_Funkcny test B - porucha vysunutia hornych kontaktov !!!
      Code = 423
      Behavior = PersistentAlarm
    [273]:
      Name = A424
      Message = ST_Funkcny test B - porucha zasunutia hornych kontaktov !!!
      Code = 424
      Behavior = PersistentAlarm
    [274]:
      Name = A425
      Message = ST_Funkcny test B - porucha vysunutia spodnych kontaktov !!!
      Code = 425
      Behavior = PersistentAlarm
    [275]:
      Name = A426
      Message = ST_Funkcny test B - porucha zasunutia spodnych kontaktov !!!
      Code = 426
      Behavior = PersistentAlarm
    [276]:
      Name = A427
      Message = ST_Funkcny test A - porucha precitania kodu paletky !!!
      Code = 427
      Behavior = PersistentAlarm
    [277]:
      Name = A428
      Message = Pracovisko 4 - Modul DI41 nieje online !!!
      Code = 428
      Behavior = PersistentAlarm
    [278]:
      Name = A429
      Message = ST_Funkcny test B - porucha precitania kodu paletky !!!
      Code = 429
      Behavior = PersistentAlarm
    [279]:
      Name = A430
      Message = Pracovisko 4 - Prekrocena teplota motora zadneho vrchneho dopravnika !!!
      Code = 430
      Behavior = PersistentAlarm
    [280]:
      Name = A431
      Message = ST9_Etiketovacka - porucha vytlacenie etikety !!!
      Code = 431
      Behavior = PersistentAlarm
    [281]:
      Name = A432
      Message = ST9_Etiketovacka - pritlak pasky v tlaciarni je odisteny !!!
      Code = 432
      Behavior = PersistentAlarm
    [282]:
      Name = A433
      Message = ST9_Etiketovacka - CAM 14 porucha komunikacie FTP !!!
      Code = 433
      Behavior = PersistentAlarm
    [283]:
      Name = A434
      Message = ST9_Etiketovacka - CAM 15 porucha komunikacie FTP !!!
      Code = 434
      Behavior = PersistentAlarm
    [284]:
      Name = A435
      Message = Pracovisko 4 - Prekrocena teplota motora priecneho dopravnika !!!
      Code = 435
      Behavior = PersistentAlarm
    [285]:
      Name = A436
      Message = Pracovisko 4 - Modul DS41 nieje online !!!
      Code = 436
    [286]:
      Name = A437
      Message = ST_Funkcny test A - je zalozeny nespravny typ spodneho kopita !!!
      Code = 437
      Behavior = PersistentAlarm
    [287]:
      Name = A438
      Message = ST_Funkcny test B - je zalozeny nespravny typ spodneho kopita !!!
      Code = 438
      Behavior = PersistentAlarm
    [288]:
      Name = A439
      Message = Pracovisko 4 - Modul DS42 nieje online !!!
      Code = 439
      Behavior = PersistentAlarm
    [289]:
      Name = A440
      Message = Pracovisko 4 - Modul SI41 nieje online !!!
      Code = 440
      Behavior = PersistentAlarm
    [290]:
      Name = A441
      Message = Pracovisko 4 - Modul SI42 nieje online !!!
      Code = 441
      Behavior = PersistentAlarm
    [291]:
      Name = A442
      Message = ST10_Vytah - porucha serva zdvihu vytahu !!!
      Code = 442
      Behavior = PersistentAlarm
    [292]:
      Name = A443
      Message = Pracovisko 4 - Prekrocena teplota motora predneho vrchneho dopravnika !!!
      Code = 443
      Behavior = PersistentAlarm
    [293]:
      Name = A444
      Message = Pracovisko 4 - Prekrocena teplota motora spodneho dopravnika !!!
      Code = 444
      Behavior = PersistentAlarm
    [294]:
      Name = A445
      Message = ST10_Vytah - Prekrocena teplota motora dopravnika !!!
      Code = 445
      Behavior = PersistentAlarm
    [295]:
      Name = A446
      Message = Pracovisko 4 - Narusenie optickej bariery na vstupe !!!
      Code = 446
      Behavior = PersistentAlarm
    [296]:
      Name = A447
      Message = Pracovisko 4 - Narusenie optickej bariery na vystupe !!!
      Code = 447
      Behavior = PersistentAlarm
    [297]:
      Name = A448
      Message = Pracovisko 4 - Bolo stlacene tlacitko CS na ovladacom paneli !!!
      Code = 448
      Behavior = PersistentAlarm
    [298]:
      Name = A449
      Message = Pracovisko 4 - Bolo stlacene tlacitko CS na rozvodnej skrini !!!
      Code = 449
      Behavior = PersistentAlarm
    [299]:
      Name = A450
      Message = ST_Funkcny test A - Porucha vyvezenia paletky zo stopra !!!
      Code = 450
      Behavior = PersistentAlarm
    [300]:
      Name = A451
      Message = ST_Funkcny test B - Porucha vyvezenia paletky zo stopra !!!
      Code = 451
      Behavior = PersistentAlarm
    [301]:
      Name = A452
      Message = ST9_Etiketovacka - Porucha vyvezenia paletky zo stopra !!!
      Code = 452
      Behavior = PersistentAlarm
    [302]:
      Name = A453
      Message = ST9_Etiketovacka - Porucha komunikacie s kamerou CAM 14 !!!
      Code = 453
      Behavior = PersistentAlarm
    [303]:
      Name = A454
      Message = ST9_Etiketovacka - Porucha komunikacie s kamerou CAM 15 !!!
      Code = 454
      Behavior = PersistentAlarm
    [304]:
      Name = A455
      Message = ST10_Vytah - Porucha komunikacie s kamerou CAM 16 !!!
      Code = 455
      Behavior = PersistentAlarm
    [305]:
      Name = A456
      Message = P4_Zdvizka za Funkcnym Testom A - Porucha vysunutia zdvizky !!!
      Code = 456
      Behavior = PersistentAlarm
    [306]:
      Name = A457
      Message = P4_Zdvizka za Funkcnym Testom A - Porucha zasunutia zdvizky !!!
      Code = 457
      Behavior = PersistentAlarm
    [307]:
      Name = A458
      Message = P4_Zdvizka za Funkcnym Testom A - Porucha strednej polohy zdvizky !!!
      Code = 458
      Behavior = PersistentAlarm
    [308]:
      Name = A459
      Message = P4_Zdvizka za Funkcnym Testom B - Porucha vysunutia zdvizky !!!
      Code = 459
      Behavior = PersistentAlarm
    [309]:
      Name = A460
      Message = P4_Zdvizka za Funkcnym Testom B - Porucha zasunutia zdvizky !!!
      Code = 460
      Behavior = PersistentAlarm
    [310]:
      Name = A461
      Message = P4_Zdvizka za Funkcnym Testom B - Porucha strednej polohy zdvizky !!!
      Code = 461
      Behavior = PersistentAlarm
    [311]:
      Name = A462
      Message = ST9_Etiketovacka - Porucha otocenia aplikatora vpred !!!
      Code = 462
      Behavior = PersistentAlarm
    [312]:
      Name = A463
      Message = ST9_Etiketovacka - Porucha otocenia aplikatora vzad !!!
      Code = 463
      Behavior = PersistentAlarm
```

### Config_5.mprecipexml - 5PC900_TS17_00/mappServices/Config_5.mprecipexml
```
Element gUserXml (Type=mprecipexml)
```

## Logical view

Binary libraries used (declarations not repeated): RUNTIME, OPERATOR, AsIecCon, astime, standard, AsBrStr, sys_lib, AsZip, AsUSB, dvframe, AsTCP, asstring, MpAlarmX 5.17.0, MpBase 5.17.0, MpRecipe 5.17.0, MpServer 5.17.0, AsICMP, FileIO, CoTrace 5.15.0
